FUNCTION_BLOCK ROBOTA1FB (* JADE WORKER *)
  (* Standard: 61499-1 *)
  (* Version 1.0, 2014-04-22, Ahmed, Fraunhofer IGD *)
  (* Compiler header: package fb.rt; *)
  (* Compiler Java Sun JDK 1.5.0 *)
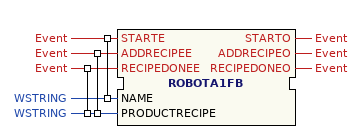
  EVENT_INPUT
    STARTE WITH NAME; (* Normal Execution Request *)
    ADDRECIPEE WITH PRODUCTRECIPE;
    RECIPEDONEE WITH PRODUCTRECIPE;
  END_EVENT
  EVENT_OUTPUT
    STARTO; (* Execution Confirmation *)
    ADDRECIPEO;
    RECIPEDONEO;
  END_EVENT
  VAR_INPUT
    NAME : WSTRING;
    PRODUCTRECIPE : WSTRING;
  END_VAR
END_FUNCTION_BLOCK
